// Mitsubishi GX Works2 project: StructuredText1   PLC: Q03UDV

PROGRAM MAIN
VAR
  Input1 : BOOL;
END_VAR
IF Input1 THEN
	Y20 := TRUE;
ELSE
	Y20 := FALSE;
END_IF;
END_PROGRAM
